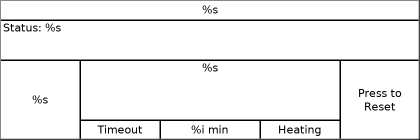
VISUALIZATION UI_Room  // 420x140
VAR_IN_OUT
	ctx			: Room_Ctx;
END_VAR
    Rectangle (0,0 420x20), "%s", text variable: CONCAT('Room ', UDINT_TO_STRING(ctx.hmi.nId))
    Rectangle (0,20 420x40), "Status: %s", text variable: ctx.hmi.sStatusText
        p55702900: ctx.hmi.nStatusColor
    Rectangle (0,60 80x80), "%s", text variable: ctx.hmi.sDisableText
        toggle ctx.hmi.bDisable
    Rectangle (340,60 80x80), "Press to Reset", invisible if: ctx.hmi.bHideReset
        toggle ctx.hmi.bReset
    Rectangle (80,60 260x60), "%s", text variable: ctx.hmi.sData
    Rectangle (160,120 100x20), "%i min", text variable: ctx.hmi.nTimeout
        OnMouseClick: write the text variable via Default
    Rectangle (80,120 80x20), "Timeout"
    Rectangle (260,120 80x20), "Heating", colour toggle: ctx.io.bValvesOpen
END_VISUALIZATION

(* stored: Version 1.1.0.1
   Visu UI_Room: Id {c568871d-7da9-43be-9c34-308759e688ca} *)
